// TIA Portal V20 export
FUNCTION_BLOCK "FB_NEW"   // FB2, LAD
{ S7_Optimized_Access := 'TRUE' }
// stored: MemoryReserve 100, SetENOAutomatically false
   VAR_INPUT
      in : Bool;
   END_VAR
   VAR_OUTPUT
      out : Bool;
   END_VAR
BEGIN

REGION Network 1
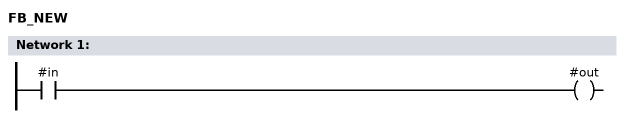
   RUNG wire#powerrail
      Contact( #in )
      Coil( #out )
   END_RUNG
   // the same network as SCL:
   #out := #in;
END_REGION
END_FUNCTION_BLOCK
